FUNCTION_BLOCK FB_ProBoxElementShuttleForksEmulation EXTENDS FB_ElementConvEmulation
(**************************************************************************************
 * 	Application		:	BoxControl Framework
 *	Revision		:	$Revision:  $
 *	Revision date	:	$Date: $
 *	Last changed by	:	$Author: $
 *	URL				:	$URL: $
 *
 *	Purpose			:	Shuttle Emulation element.
 *
 * ------------------------------------------------------------------------------------
 *	Copyright Swisslog [IP AG], Switzerland. All rights reserved.
 * 
 * ------------------------------------------------------------------------------------
 *	
 * 	Revision History: 
 *
 * 	VERSION			DATE			INITIALS			DESCRIPTION
 *
 **************************************************************************************)
 VAR_INPUT
 		
END_VAR
VAR
	pElement						: POINTER TO FB_ProBoxElementShuttleForks; // Address to element
	rElement						: REFERENCE TO FB_ProBoxElementShuttleForks; // Reference to element
	j : INT;	
	DbgHwInputElShuttle 			: ST_HW_InputsProBoxElementShuttleForks;//ST_HW_InputsShuttle;
	
	Debug:BOOL;
END_VAR

(**************************************************************************************************************
   Initialization
***************************************************************************************************************)
A_Init();

(**************************************************************************************************************
   Update reference
***************************************************************************************************************)
A_UpdateReference();

(**************************************************************************************************************
   Emulation
***************************************************************************************************************)
// If emulation element is initialized
IF ElementData.Init THEN
	
	// Update real data
	M_UpdateRealObjectData();	

	//Set emulation speed	
	rElement.P_EmuSpeed	:= ProBoxSystem.EMULATION_SPEED;
		
	// Overwrite inputs
	_M_OverWriteInputs();

END_IF

METHOD PRIVATE _M_OverWriteInputs : BOOL
VAR_INPUT
END_VAR
VAR
	i : INT;
	FunctionNoConvA 				: E_FunctionNumber;
	FunctionNoConvB 				: E_FunctionNumber;	
	NumberOfZonesConvA				: INT:=1;
	NumberOfZonesConvB				: INT:=1;
	
	DriveA_Run_12					: BOOL;	//Conveyor A FWD
	DriveA_Run_21					: BOOL; //Conveyor A RWD
	DriveB_Run_12					: BOOL; //Conveyor B FWD
	DriveB_Run_21					: BOOL; //Conveyor B RWD
END_VAR
//Get the function number of the shuttle car conveyor A and B
//Get the function number of the vertical lift conveyor A and B
IF(__ISVALIDREF(ElementRegistry[rElement.ConfigElement.eElementNumber].rElementData)) THEN
	FunctionNoConvA:= ElementRegistry[rElement.ConfigElement.eElementNumber].rElementData.MemberList.FunctionList[1].eFunctionNumber;
	FunctionNoConvB:= ElementRegistry[rElement.ConfigElement.eElementNumber].rElementData.MemberList.FunctionList[2].eFunctionNumber;
ELSE
	RETURN; //error
END_IF

IF(__ISVALIDREF(FunctionRegistry[FunctionNoConvA].rSettingsFunction)) THEN
	NumberOfZonesConvA := FunctionRegistry[FunctionNoConvA].rSettingsFunction.NumberOfZones;
END_IF
IF(__ISVALIDREF(FunctionRegistry[FunctionNoConvB].rSettingsFunction)) THEN
	NumberOfZonesConvB := FunctionRegistry[FunctionNoConvB].rSettingsFunction.NumberOfZones;
END_IF



IF(ElementData.Init AND NOT Debug) THEN
	

	//set temp variables
	DriveA_Run_12 := ElementRegistry[rElement.ConfigElement.eElementNumber].rElementData.FunctionOrder.ReqDriveRun AND ElementRegistry[rElement.ConfigElement.eElementNumber].rElementData.FunctionOrder.ReqDriveDirection;
	DriveA_Run_21 := ElementRegistry[rElement.ConfigElement.eElementNumber].rElementData.FunctionOrder.ReqDriveRun AND NOT ElementRegistry[rElement.ConfigElement.eElementNumber].rElementData.FunctionOrder.ReqDriveDirection;
	DriveB_Run_12:= ElementRegistry[rElement.ConfigElement.eElementNumber].rElementData.FunctionOrder.ReqDriveRun_34 AND ElementRegistry[rElement.ConfigElement.eElementNumber].rElementData.FunctionOrder.ReqDriveDirection_34;
	DriveB_Run_21:= ElementRegistry[rElement.ConfigElement.eElementNumber].rElementData.FunctionOrder.ReqDriveRun_34 AND NOT ElementRegistry[rElement.ConfigElement.eElementNumber].rElementData.FunctionOrder.ReqDriveDirection_34;

	
	
	F_MPD_GetOverhangSensorStatus(
			MPD_Function:= FunctionNoConvA,  // Conveyor A
			ZonesPerFunction:= NumberOfZonesConvA,
			Drive_Run_12:= DriveA_Run_12, //rElement.HW_Outputs.DriveCV_A.Drive_Run_12,
			Drive_Run_21:= DriveA_Run_21,//rElement.HW_Outputs.DriveCV_A.Drive_Run_21,
			SensorOverhang12=>rElement.HW_Inputs.Conv.SensorOverhangLeft,
			SensorOverhang21=>rElement.HW_Inputs.Conv.SensorOverhangRight);
	
	
	

	//Set overhang sensor value on adjacent functions
	//simulate Sensor overhang is activated during transfer
	FOR i := 1 TO GVL_MPD.MAXPDs BY 1 DO	
		IF  rElement.Config.ConvCFG[i].eFunctionNumber <> E_FunctionNumber.F_BEGIN_FUNCTION THEN
			rElement.M_SetOverhangSensor(
				eFunctionnumber:= rElement.Config.ConvCFG[i].eFunctionNumber,			
				SensorValue:= NOT (F_PB_GetTransportControlDataRef(rElement.Config.ConvCFG[i].eFunctionNumber,1).DriveRunning AND 
								  (DriveA_Run_12 OR DriveA_Run_21 OR DriveB_Run_12 OR DriveB_Run_21)));
						
		ELSE
			EXIT;
		END_IF
	END_FOR
	
	//Set other element HW input
	rElement.HW_Inputs.MotorUnitOK 	:= DbgHwInputElShuttle.MotorUnitOK;
	rElement.HW_Inputs.EndLimit		:= DbgHwInputElShuttle.EndLimit;
			
END_IF
END_METHOD

ACTION A_Init:
(**************************************************************************************
 * 	NAME		A_Init
 * 	FUNCTION	Initialize emulated dummy element
 **************************************************************************************)

// If element is not initialized
IF NOT ElementData.Init THEN

	// Check that linked element number is valid
	IF eElementNumber > E_ElementNumber.E_BEGIN_ELEMENT AND
	   eElementNumber < E_ElementNumber.E_END_ELEMENT THEN
		
			// Check that the real module is initialized
			IF F_IsElementInitialized(eElementNumber) THEN
				// Module is initialized
				ElementData.Init := TRUE;
				
				// Send debug message
				DebugMsg := CONCAT('Initialization done. Element: ', ElementRegistry[eElementNumber].ElementName);
				fbDebugMsg.M_SendInfoMsg(DebugMsg);
				
				// Initialize real module
				F_InitializeElement(eElementNumber := eElementNumber);
			END_IF
	END_IF
END_IF
END_ACTION

ACTION A_UpdateReference:
(**************************************************************************************
 * 	NAME		A_UpdateReference
 * 	FUNCTION	Update reference to real object
 **************************************************************************************)

// Check valid element number
IF eElementNumber > E_ElementNumber.E_BEGIN_ELEMENT AND
   eElementNumber < E_ElementNumber.E_END_ELEMENT THEN

	// Is reference valid  
	IF __ISVALIDREF(ElementRegistry[eElementNumber].rElement) THEN
		// Build address to reference
		pElement := ADR(ElementRegistry[eElementNumber].rElement);

		// If address is possible
		IF pElement <> 0 THEN
			// Build reference to memory
			rElement REF= pElement^;
		ELSE
			// Reinitialize module
			ElementData.Init := FALSE;
		END_IF
	ELSE
		// Reinitialize module
		ElementData.Init := FALSE;
	END_IF
END_IF
END_ACTION

METHOD FB_init : BOOL
VAR_INPUT
	bInitRetains : BOOL; // if TRUE, the retain variables are initialized (warm start / cold start)
	bInCopyCode : BOOL;  // if TRUE, the instance afterwards gets moved into the copy code (online change)
END_VAR
VAR
	i:INT;
END_VAR
IF(bInitRetains OR bInCopyCode) THEN
	
	DbgHwInputElShuttle.MotorUnitOK :=  TRUE;	
	DbgHwInputElShuttle.EndLimit := TRUE;
END_IF
END_METHOD

END_FUNCTION_BLOCK

(* stored: Version 1.1.0.1, ProductVersion 3.1.4024.9
   POU FB_ProBoxElementShuttleForksEmulation: Id {019b56da-3c3e-4a9b-bedf-3ef4119eaddf}, SpecialFunc None
   Method _M_OverWriteInputs: Id {0c388537-48ba-459d-8457-b8bbb27872cc}
   Action A_Init: Id {d1c93436-50fe-452c-9554-4b5b5dd08662}
   Action A_UpdateReference: Id {f976d342-4fba-49e6-9d00-3cf9d419af7f}
   Method FB_init: Id {d09cc962-ff41-4e5d-b912-51ed406ddb56} *)
